// TIA Portal V16 export
// export: Created 2023-01-04T15:44:05.2202127Z, ExportSetting WithDefaults, DisplayName Totally Integrated Automation Portal, DisplayVersion V16, DisplayName TIA Portal Version Control Interface, DisplayVersion V16, DisplayName TIA Portal Openness, DisplayVersion V16, DisplayName STEP 7 Professional, DisplayVersion V16, DisplayName STEP 7 Safety, DisplayVersion V16, DisplayName WinCC Advanced, DisplayVersion V16
ORGANIZATION_BLOCK "Main"   // OB1, LAD, ProgramCycle
TITLE = "Main Program Sweep (Cycle)"
{ S7_Optimized_Access := 'TRUE' }
VERSION : 0.1
// stored: AutoNumber true, IsIECCheckEnabled false, SetENOAutomatically false
   VAR_INPUT
      Initial_Call : Bool;   // Initial call of this OB
      Remanence : Bool;   // =True, if remanent data are available
   END_VAR
   VAR_TEMP   // added for the SCL form of the ladder/FBD networks
      _w1 : Bool;
      _w2 : Bool;
   END_VAR
BEGIN

REGION Network 1: Tank 1 and Tank 2 re-filling Logic
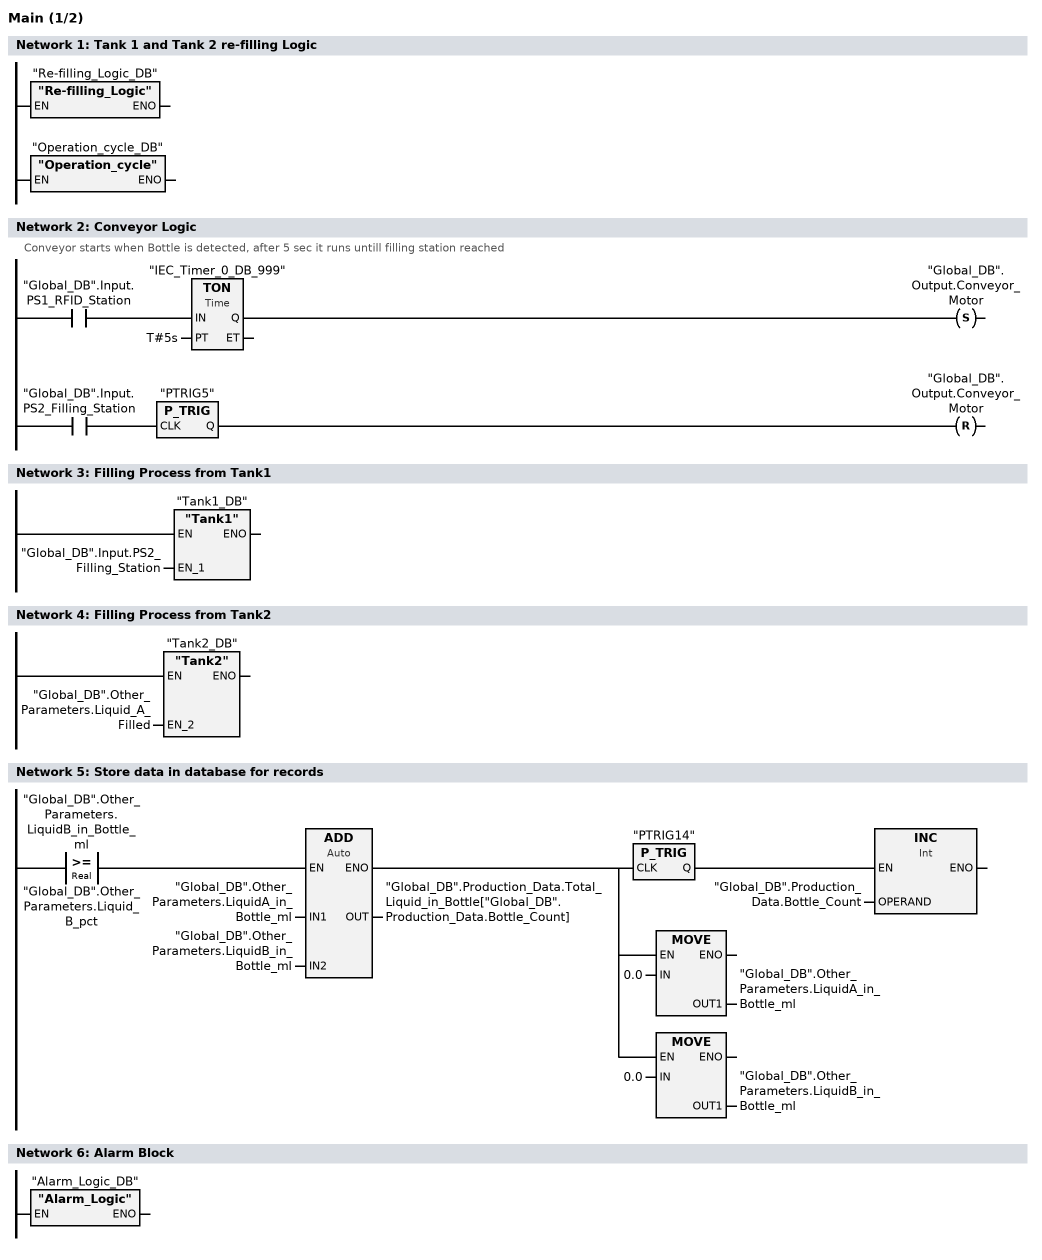
   RUNG wire#powerrail
      "Re-filling_Logic_DB"()
   END_RUNG
   RUNG wire#powerrail
      "Operation_cycle_DB"()
   END_RUNG
   // the same network as SCL:
   "Re-filling_Logic_DB"();   // "Re-filling_Logic"
   "Operation_cycle_DB"();   // "Operation_cycle"
END_REGION

REGION Network 2: Conveyor Logic
   // Conveyor starts when Bottle is detected, after 5 sec it runs untill filling station reached
   RUNG wire#powerrail
      Contact( "Global_DB".Input.PS1_RFID_Station )
      { S7_Templates := "time_type := Time" } "IEC_Timer_0_DB_999".TON(pt := T#5s, et =>)
      S_Coil( "Global_DB".Output.Conveyor_Motor )
   END_RUNG
   RUNG wire#powerrail
      Contact( "Global_DB".Input.PS2_Filling_Station )
      P_Trig( "PTRIG5" )
      R_Coil( "Global_DB".Output.Conveyor_Motor )
   END_RUNG
   // the same network as SCL:
   "IEC_Timer_0_DB_999".TON(IN := "Global_DB".Input.PS1_RFID_Station, PT := T#5s);
   IF "IEC_Timer_0_DB_999".Q THEN "Global_DB".Output.Conveyor_Motor := TRUE; END_IF;
   #_w1 := "Global_DB".Input.PS2_Filling_Station AND NOT "PTRIG5";   // rising edge
   "PTRIG5" := "Global_DB".Input.PS2_Filling_Station;
   IF #_w1 THEN "Global_DB".Output.Conveyor_Motor := FALSE; END_IF;
END_REGION

REGION Network 3: Filling Process from Tank1
   RUNG wire#powerrail
      "Tank1_DB"(EN_1 := "Global_DB".Input.PS2_Filling_Station)
   END_RUNG
   // the same network as SCL:
   "Tank1_DB"(EN_1 := "Global_DB".Input.PS2_Filling_Station);   // "Tank1"
END_REGION

REGION Network 4: Filling Process from Tank2
   RUNG wire#powerrail
      "Tank2_DB"(EN_2 := "Global_DB".Other_Parameters.Liquid_A_Filled)
   END_RUNG
   // the same network as SCL:
   "Tank2_DB"(EN_2 := "Global_DB".Other_Parameters.Liquid_A_Filled);   // "Tank2"
END_REGION

REGION Network 5: Store data in database for records
   RUNG wire#powerrail
      { S7_Templates := "SrcType := Real" } GE_Contact(in1 := "Global_DB".Other_Parameters.LiquidB_in_Bottle_ml, in2 := "Global_DB".Other_Parameters.Liquid_B_pct)
      Add(in1 := "Global_DB".Other_Parameters.LiquidA_in_Bottle_ml, in2 := "Global_DB".Other_Parameters.LiquidB_in_Bottle_ml, out => "Global_DB".Production_Data.Total_Liquid_in_Bottle["Global_DB".Production_Data.Bottle_Count])
      wire#w1
      P_Trig( "PTRIG14" )
      { S7_Templates := "DestType := Int" } Inc( "Global_DB".Production_Data.Bottle_Count )
   END_RUNG
   RUNG wire#w1
      Move(in := 0.0, out1 => "Global_DB".Other_Parameters.LiquidA_in_Bottle_ml)
   END_RUNG
   RUNG wire#w1
      Move(in := 0.0, out1 => "Global_DB".Other_Parameters.LiquidB_in_Bottle_ml)
   END_RUNG
   // the same network as SCL:
   #_w1 := "Global_DB".Other_Parameters.LiquidB_in_Bottle_ml >= "Global_DB".Other_Parameters.Liquid_B_pct;
   IF #_w1 THEN
       "Global_DB".Production_Data.Total_Liquid_in_Bottle["Global_DB".Production_Data.Bottle_Count] := "Global_DB".Other_Parameters.LiquidA_in_Bottle_ml + "Global_DB".Other_Parameters.LiquidB_in_Bottle_ml;
   END_IF;
   #_w2 := #_w1 AND NOT "PTRIG14";   // rising edge
   "PTRIG14" := #_w1;
   IF #_w2 THEN
       "Global_DB".Production_Data.Bottle_Count := "Global_DB".Production_Data.Bottle_Count + 1;
   END_IF;
   IF #_w1 THEN
       "Global_DB".Other_Parameters.LiquidA_in_Bottle_ml := 0.0;
       "Global_DB".Other_Parameters.LiquidB_in_Bottle_ml := 0.0;
   END_IF;
END_REGION

REGION Network 6: Alarm Block
   RUNG wire#powerrail
      "Alarm_Logic_DB"()
   END_RUNG
   // the same network as SCL:
   "Alarm_Logic_DB"();   // "Alarm_Logic"
END_REGION

REGION Network 7: Process after bottle is filled
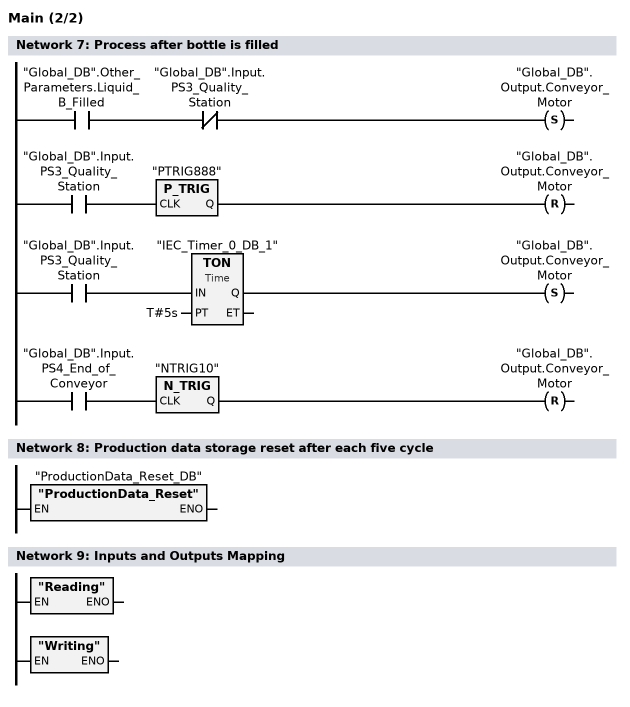
   RUNG wire#powerrail
      Contact( "Global_DB".Other_Parameters.Liquid_B_Filled )
      I_Contact( "Global_DB".Input.PS3_Quality_Station )
      S_Coil( "Global_DB".Output.Conveyor_Motor )
   END_RUNG
   RUNG wire#powerrail
      Contact( "Global_DB".Input.PS3_Quality_Station )
      P_Trig( "PTRIG888" )
      R_Coil( "Global_DB".Output.Conveyor_Motor )
   END_RUNG
   RUNG wire#powerrail
      Contact( "Global_DB".Input.PS3_Quality_Station )
      { S7_Templates := "time_type := Time" } "IEC_Timer_0_DB_1".TON(pt := T#5s, et =>)
      S_Coil( "Global_DB".Output.Conveyor_Motor )
   END_RUNG
   RUNG wire#powerrail
      Contact( "Global_DB".Input.PS4_End_of_Conveyor )
      N_Trig( "NTRIG10" )
      R_Coil( "Global_DB".Output.Conveyor_Motor )
   END_RUNG
   // the same network as SCL:
   IF "Global_DB".Other_Parameters.Liquid_B_Filled AND NOT "Global_DB".Input.PS3_Quality_Station THEN
       "Global_DB".Output.Conveyor_Motor := TRUE;
   END_IF;
   #_w1 := "Global_DB".Input.PS3_Quality_Station AND NOT "PTRIG888";   // rising edge
   "PTRIG888" := "Global_DB".Input.PS3_Quality_Station;
   IF #_w1 THEN "Global_DB".Output.Conveyor_Motor := FALSE; END_IF;
   "IEC_Timer_0_DB_1".TON(IN := "Global_DB".Input.PS3_Quality_Station, PT := T#5s);
   IF "IEC_Timer_0_DB_1".Q THEN "Global_DB".Output.Conveyor_Motor := TRUE; END_IF;
   #_w2 := NOT "Global_DB".Input.PS4_End_of_Conveyor AND "NTRIG10";   // falling edge
   "NTRIG10" := "Global_DB".Input.PS4_End_of_Conveyor;
   IF #_w2 THEN "Global_DB".Output.Conveyor_Motor := FALSE; END_IF;
END_REGION

REGION Network 8: Production data storage reset after each five cycle
   RUNG wire#powerrail
      "ProductionData_Reset_DB"()
   END_RUNG
   // the same network as SCL:
   "ProductionData_Reset_DB"();   // "ProductionData_Reset"
END_REGION

REGION Network 9: Inputs and Outputs Mapping
   RUNG wire#powerrail
      "Reading"()
   END_RUNG
   RUNG wire#powerrail
      "Writing"()
   END_RUNG
   // the same network as SCL:
   "Reading"();
   "Writing"();
END_REGION
END_ORGANIZATION_BLOCK
